Staubli VAL3: clkGlueGlass.pgx

program clkGlueGlass()
begin
  bGlueGlass=true
end
